// TIA Portal V18 export
// export: Created 2026-06-08T16:08:49.9609628Z, ExportSetting WithDefaults, DisplayName Totally Integrated Automation Portal, DisplayVersion V18, DisplayName TIA Portal Openness, DisplayVersion V18, DisplayName TIA Portal Version Control Interface, DisplayVersion V18, DisplayName STEP 7 Professional, DisplayVersion V18, DisplayName STEP 7 Safety, DisplayVersion V18, DisplayName WinCC Professional, DisplayVersion V18
ORGANIZATION_BLOCK "Cyclic interrupt"   // OB30, LAD, CyclicInterrupt
{ S7_Optimized_Access := 'TRUE' }
VERSION : 0.1
// stored: AutoNumber true, IsIECCheckEnabled false, SetENOAutomatically false
   VAR_INPUT
      Initial_Call : Bool;   // Initial call of this OB
      Event_Count : Int;   // Events discarded
   END_VAR
BEGIN

REGION Network 1
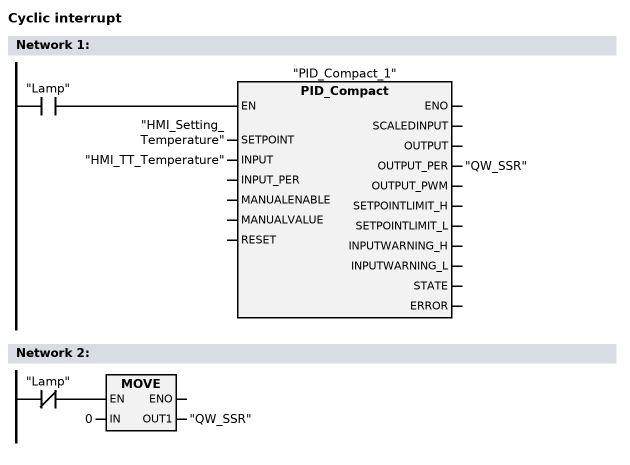
   RUNG wire#powerrail
      Contact( "Lamp" )
      "PID_Compact_1".PID_Compact(Setpoint := "HMI_Setting_Temperature", Input := "HMI_TT_Temperature", Input_PER :=, ManualEnable :=, ManualValue :=, Reset :=, ScaledInput =>, Output =>, Output_PER => "QW_SSR", Output_PWM =>, SetpointLimit_H =>, SetpointLimit_L =>, InputWarning_H =>, InputWarning_L =>, State =>, Error =>)
   END_RUNG
   // the same network as SCL:
   IF "Lamp" THEN
       "PID_Compact_1"(Setpoint := "HMI_Setting_Temperature", Input := "HMI_TT_Temperature", Output_PER => "QW_SSR");   // PID_Compact
   END_IF;
END_REGION

REGION Network 2
   RUNG wire#powerrail
      I_Contact( "Lamp" )
      Move(in := 0, out1 => "QW_SSR")
   END_RUNG
   // the same network as SCL:
   IF NOT "Lamp" THEN "QW_SSR" := 0; END_IF;
END_REGION
END_ORGANIZATION_BLOCK
